// SIMATIC S7-200 project (STEP 7-Micro/WIN), CPU 221 REL 01.10

SYMBOL_TABLE USER1
A1               I0.0
B                I0.1
C                I0.2
D                I0.3
X                Q0.0
Y                Q0.1
L                Q0.2
P                Q0.3
T                Q0.4
M                M0.1
END_SYMBOL_TABLE

ORGANIZATION_BLOCK MAIN:OB1
TITLE=PROGRAM COMMENTS
BEGIN
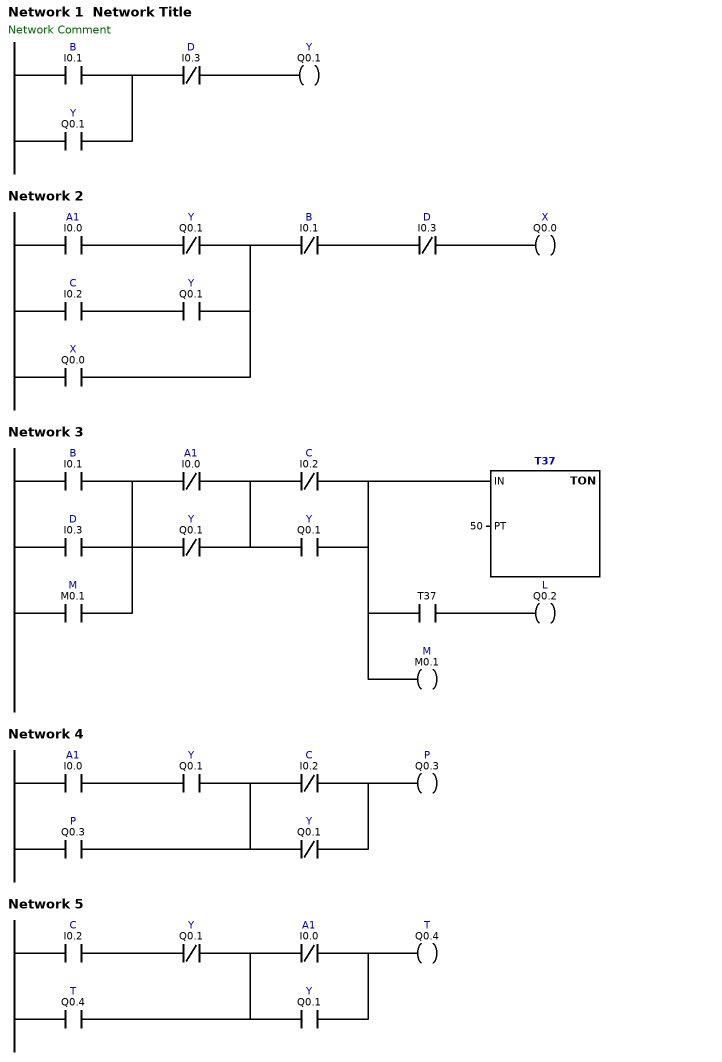
Network 1 // Network Title
// Network Comment
LD     B:I0.1
O      Y:Q0.1
AN     D:I0.3
=      Y:Q0.1
Network 2
LD     A1:I0.0
AN     Y:Q0.1
LD     C:I0.2
A      Y:Q0.1
OLD
O      X:Q0.0
AN     B:I0.1
AN     D:I0.3
=      X:Q0.0
Network 3
LD     B:I0.1
O      D:I0.3
O      M:M0.1
LDN    A1:I0.0
ON     Y:Q0.1
ALD
LDN    C:I0.2
O      Y:Q0.1
ALD
LPS
TON    T37, 50
A      T37
=      L:Q0.2
LPP
=      M:M0.1
Network 4
LD     A1:I0.0
A      Y:Q0.1
O      P:Q0.3
LDN    C:I0.2
ON     Y:Q0.1
ALD
=      P:Q0.3
Network 5
LD     C:I0.2
AN     Y:Q0.1
O      T:Q0.4
LDN    A1:I0.0
O      Y:Q0.1
ALD
=      T:Q0.4
END_ORGANIZATION_BLOCK
